// TIA Portal V19 export
DATA_BLOCK "ProductionMng"   // DB169
// stored: InstanceOfName ProductionMng_FB, InstanceOfType FB
"ProductionMng_FB"
   // VAR_INPUT
   //    Cin : "Prod_CIn";
   // END_VAR
   // VAR_OUTPUT
   //    COut : "Prod_COut";
   // END_VAR
   // VAR_IN_OUT
   //    Pers : "Prod_Pers";
   // END_VAR
   // VAR
   //    Warnings : Struct
   //       Error_Send_Message_To_MES_Cumulative : Bool;
   //       SetUp { ExternalAccessible := 'False'; ExternalVisible := 'False'; ExternalWritable := 'False'} : Struct
   //          PUSH_MSG101 : "MES_Err_&_Msg";
   //          Caricamento_PPrf : Struct
   //             Err_Load_PPrf : Bool;
   //             Err_Load_Timeout : Bool;
   //             Err_NumeroProgrammaNonValido : Bool;
   //             Err_NonCorrisponde_W_A : Bool;
   //             Err_NonCorrisponde_H_B : Bool;
   //             Err_NonCorrisponde_Spessore : Bool;
   //          END_STRUCT;
   //          Attesa_Avvio_SetUp_Automatico : Bool;
   //          SetUp_Automatico_Avviato : Bool;
   //          Attesa_Completamento_SetUp_Manuale : Bool;
   //          Attesa_Inizio_Inserimento_lamiera : Bool;
   //          Attesa_Fine_inserimento_lamiera : Bool;
   //          Attesa_Taglio_di_Intestazione : Bool;
   //          PUSH_MSG102 : "MES_Err_&_Msg";
   //       END_STRUCT;
   //       Error_Pop_O_ACT_to_O_ENDING : "MES_Err";
   //       Error_Pop_O_TODO_to_O_ACT : "MES_Err";
   //       O_ACT_Empty : Bool;
   //    END_STRUCT;
   //    Messages : Struct
   //       Err_MSG131_Part_GOOD : "MES_Err_&_Msg";
   //       Err_MSG131_Part_NG { S7_SetPoint := 'True'} : "MES_Err_&_Msg";
   //       Err_MSG131_Part_GOOD_R : "MES_Err_&_Msg";
   //       Err_MSG131_Part_NG_R { S7_SetPoint := 'True'} : "MES_Err_&_Msg";
   //       Err_MSG131_Part_DELETE { S7_SetPoint := 'True'} : "MES_Err_&_Msg";
   //       Err_MSG131_Beam_GOOD : "MES_Err_&_Msg";
   //       Err_MSG131_Beam_GOOD_R : "MES_Err_&_Msg";
   //       Err_MSG131_Beam_NG_R : "MES_Err_&_Msg";
   //       Err_MSG131_Beam_DELETE : "MES_Err_&_Msg";
   //       Err_MSG131_O_ACT_Status_Update { S7_SetPoint := 'True'} : "MES_Err_&_Msg";
   //       Err_MSG131_O_TODO_Status_Update { S7_SetPoint := 'True'} : "MES_Err_&_Msg";
   //       Err_MSG131_O_ENDING_Status_Update { S7_SetPoint := 'True'} : "MES_Err_&_Msg";
   //       Err_MSG131_O_OUT_Status_Update { S7_SetPoint := 'True'} : "MES_Err_&_Msg";
   //       Err_Msg201 { ExternalAccessible := 'False'; ExternalVisible := 'False'; ExternalWritable := 'False'} : "MES_Err_&_Msg";
   //       Err_Msg211 { ExternalAccessible := 'False'; ExternalVisible := 'False'; ExternalWritable := 'False'} : "MES_Err_&_Msg";
   //       Err_Msg310_O_ACT { ExternalAccessible := 'False'; ExternalVisible := 'False'; ExternalWritable := 'False'} : "MES_Err_&_Msg";
   //       Err_Msg310_O_ENDING { ExternalAccessible := 'False'; ExternalVisible := 'False'; ExternalWritable := 'False'; S7_SetPoint := 'True'} : Array[1.."PROD_ENDING_ITEMS"] of "MES_Err_&_Msg";
   //       Err_Msg311_O_ACT { ExternalAccessible := 'False'; ExternalVisible := 'False'; ExternalWritable := 'False'} : "MES_Err_&_Msg";
   //       Err_Msg311_O_ENDING { ExternalAccessible := 'False'; ExternalVisible := 'False'; ExternalWritable := 'False'; S7_SetPoint := 'True'} : Array[1.."PROD_ENDING_ITEMS"] of "MES_Err_&_Msg";
   //       Err_Msg411 { ExternalAccessible := 'False'; ExternalVisible := 'False'; ExternalWritable := 'False'} : "MES_Err_&_Msg";
   //       Err_Msg413 { ExternalAccessible := 'False'; ExternalVisible := 'False'; ExternalWritable := 'False'} : "MES_Err_&_Msg";
   //       Err_Msg423 { ExternalAccessible := 'False'; ExternalVisible := 'False'; ExternalWritable := 'False'} : "MES_Err_&_Msg";
   //       Err_MSG431_Part_BAD { S7_SetPoint := 'True'} : "MES_Err_&_Msg";
   //       Err_MSG431_Part_NG { S7_SetPoint := 'True'} : "MES_Err_&_Msg";
   //       Err_MSG431_Part_NG_R { S7_SetPoint := 'True'} : "MES_Err_&_Msg";
   //       Err_MSG431_Part_DELETE { S7_SetPoint := 'True'} : "MES_Err_&_Msg";
   //       Err_MSG431_Beam_NG_R { S7_SetPoint := 'True'} : "MES_Err_&_Msg";
   //       Err_MSG431_Beam_DELETE { S7_SetPoint := 'True'} : "MES_Err_&_Msg";
   //       Err_Msg431_FineLamieraRF { S7_SetPoint := 'True'} : "MES_Err_&_Msg";
   //    END_STRUCT;
   //    i : Int;
   //    Part_Done_Event : Struct
   //       Exe_Update : Bool;
   //       ACK_Done : Bool;
   //       Is_BAD_WELD : Bool;
   //       IS_BAD_EXCEED_TOL : Bool;
   //       Is_BAD_TEST : Bool;
   //       is_GOOD : Bool;
   //       Is_TO_CHECK_LEN : Bool;
   //       OK_StampoSpessore : Bool;
   //       OK_StampoColata : Bool;
   //       Save_PTrk : "PTrk_Item";
   //       LenErr : Real;
   //       LenErrAbs : Real;
   //       LenErrBADLimit : Real;
   //       RETVAL_PTrk_Update : Int;
   //       RETVAL_Next_To_Do : Int;
   //    END_STRUCT;
   //    Part_GOOD_R_Event : Struct
   //       Exe : Bool;
   //       Save_PTrk : "PTrk_Item";
   //    END_STRUCT;
   //    Part_NG_R_Event : Struct
   //       Exe : Bool;
   //       Save_PTrk : "PTrk_Item";
   //       Indx { S7_SetPoint := 'True'} : Int;
   //    END_STRUCT;
   //    Part_Delete_Event : Struct
   //       Exe : Bool;
   //       index : Int;
   //       P_Array_Code : Int;
   //       PTrk_Save : "PTrk_Item";
   //    END_STRUCT;
   //    Beam_Done_Event : Struct
   //       GOOD : Bool;
   //       TO_CHECK : Bool;
   //    END_STRUCT;
   //    Beam_Recondition_Event : Struct
   //       GOOD_R : Bool;
   //       NG_R : Bool;
   //       NG_R_Index : Int;
   //    END_STRUCT;
   //    Beam_Delete_Event : Struct
   //       Exe : Bool;
   //       Index : Int;
   //       B_Array_Code : Int;
   //       BTRK_Item_Save : "BTrk_item";
   //    END_STRUCT;
   //    Update_Part_BAD : "Prod_O_Counters_Update_Push_MSG431_PTRK";
   //    Update_Part_GOOD : "Prod_O_Counters_Update_Part_GOOD";
   //    Update_Part_TOCHECK : "Prod_O_Counters_Update_Part_TOCHECK";
   //    Update_Part_NG : "Prod_O_Counters_Update_Part_NG";
   //    Update_Part_GOOD_R : "Prod_O_Counters_Update_Part_GOOD_R";
   //    Update_Part_NG_R : "Prod_O_Counters_Update_Part_NG_R";
   //    Update_Part_Delete : "Prod_O_Counters_Update_Part_Delete";
   //    Update_Beam_GOOD : "Prod_O_Counters_Update_Beam_GOOD";
   //    Update_Beam_GOOD_R : "Prod_O_Counters_Update_Beam_GOOD_R";
   //    Update_Beam_TOCHECK : "Prod_O_Counters_Update_Beam_TOCHECK";
   //    Update_Beam_NG_R : "Prod_O_Counters_Update_Beam_NG_R";
   //    Update_Beam_Delete : "Prod_O_Counters_Update_Beam_Delete";
   //    O_Status_Update : "Prod_O_Status_Update";
   //    Clean_O_ENDING { S7_SetPoint := 'True'} : "Prod_O_ENDING_Clean";
   //    Sospensioni { S7_SetPoint := 'True'} : "Prod_Update_Stato_Sospensioni_Mng";
   //    HMI_Mng { S7_SetPoint := 'True'} : "Prod_HMI_Mng";
   //    SetUp_Mng { S7_SetPoint := 'True'} : "Prod_SetUp_Mng_Vrs2";
   //    Stato_Pacchi { S7_SetPoint := 'True'} : "Prod_O_Update_Stato_Pacchi_Mng";
   //    Coils_Mng { S7_SetPoint := 'True'} : "Prod_Coils_Mng";
   //    OrdineKanban { S7_SetPoint := 'True'} : Bool;
   // END_VAR
BEGIN
END_DATA_BLOCK
